// TIA Portal project "Pick and Place (Basic)" (V16)
// Vorlageprojekt für das Buch mit Zielsystem S7-1200

(* hardware
DEVICE "S7-1200-Station_1"  S7-1200 Station
   slot 0: "Baugruppenträger_0"  Rack  V1.0
   slot 1: "PLC_1"  CPU 1211C DC/DC/DC  6ES7 211-1AE40-0XB0  V4.1
*)

// ===== PLC "PLC_1"  CPU 1211C DC/DC/DC =====

VAR_GLOBAL   // PLC tag table "Standard-Variablentabelle"
   "Start" AT %I10.0 : Bool;
   "Stop" AT %I10.1 : Bool;
   "Item at entry" AT %I10.2 : Bool;
   "Item at exit" AT %I10.3 : Bool;
   "Moving X" AT %I10.4 : Bool;
   "Moving Z" AT %I10.5 : Bool;
   "Item detected" AT %I10.6 : Bool;
   "X1" AT %M1.0 : Bool;
   "X2" AT %M1.1 : Bool;
   "X3" AT %M1.2 : Bool;
   "X4" AT %M1.3 : Bool;
   "X5" AT %M1.4 : Bool;
   "X6" AT %M1.5 : Bool;
   "Entry Conveyor" AT %Q10.0 : Bool;
   "Exit Conveyor" AT %Q10.1 : Bool;
   "Move X" AT %Q10.2 : Bool;
   "Move Z" AT %Q10.3 : Bool;
   "Grab" AT %Q10.4 : Bool;
   "X7" AT %M1.6 : Bool;
   "X8" AT %M1.7 : Bool;
END_VAR

// folder: System blocks/Program resources

DATA_BLOCK "T1"   // DB1
{ S7_Optimized_Access := 'TRUE' }
AUTHOR : Simatic
FAMILY : IEC
NAME : IEC_TMR
VERSION : 1.0
// stored: InstanceOfName IEC_TIMER
"IEC_TIMER"
BEGIN
END_DATA_BLOCK

DATA_BLOCK "T2"   // DB2
{ S7_Optimized_Access := 'TRUE' }
AUTHOR : Simatic
FAMILY : IEC
NAME : IEC_TMR
VERSION : 1.0
// stored: InstanceOfName IEC_TIMER
"IEC_TIMER"
BEGIN
END_DATA_BLOCK

// folder: (top level)

FUNCTION "MHJ-PLC-Lab-Function-S71200" : Void   // FC9000, SCL
{ S7_Optimized_Access := 'TRUE' }
VERSION : 0.1
   VAR_TEMP
      rdTimeReturn : Int;
      outputTime : DTL;
      SyncVal : Byte;
      forVal : Int;
      forVal_2 : Int;
      Value : Byte;
   END_VAR
   VAR CONSTANT
      CompVal : Byte := 16#34;
      Value_01 : Byte := 16#11;
      Value_01_DW : DWord := 16#A165_D992;
      Value_02_DW : DWord := 16#58BE_4401;
   END_VAR
BEGIN

   #Value:=PEEK(area := 16#82,
        dbNumber := 0,
        byteOffset := 511);
   #Value := #Value + 1;

   POKE(area := 16#82,
        dbNumber := 0,
        byteOffset := 511,
        value := #Value);

   POKE(area:=16#81,
        dbNumber:=0,
        byteOffset:=1016,
        value:=#Value_01_DW);
   POKE(area := 16#81,
        dbNumber := 0,
        byteOffset := 1020,
        value := #Value_02_DW);

   POKE(area := 16#81,
        dbNumber := 0,
        byteOffset := 511,
        value := B#16#00);

   FOR #forVal := 0 TO 120 DO
       FOR #forVal_2:=0 TO 10 DO
           #rdTimeReturn:=RD_SYS_T(#outputTime);
           #rdTimeReturn := WR_SYS_T(#outputTime);
           #rdTimeReturn := RD_SYS_T(#outputTime);
           #rdTimeReturn := WR_SYS_T(#outputTime);
       END_FOR;
       #SyncVal:= PEEK(area := 16#81,
                      dbNumber := 0,
                      byteOffset := 511);
       IF #SyncVal = #CompVal THEN
          GOTO M_1;
       END_IF;
   END_FOR;
   RETURN;

   M_1:
   POKE(area := 16#81,
        dbNumber := 0,
        byteOffset := 511,
        value := B#16#0);
END_FUNCTION

ORGANIZATION_BLOCK "Main"   // OB1, LAD, ProgramCycle
TITLE = "Main Program Sweep (Cycle)"
{ S7_Optimized_Access := 'TRUE' }
VERSION : 0.1
   VAR_INPUT
      Initial_Call : Bool;   // Initial call of this OB
      Remanence : Bool;   // =True, if remanent data are available
   END_VAR
   VAR_TEMP   // added for the SCL form of the ladder/FBD networks
      _w1 : Bool;
   END_VAR
BEGIN

REGION Network 1: Konnektierungsbaustein für PLC-Lab
   // Im Netzwerk 1 wird der Konnektierungsbaustein für PLC-Lab aufgerufen.
   // Dieser Aufruf darf nicht entfernt werden!
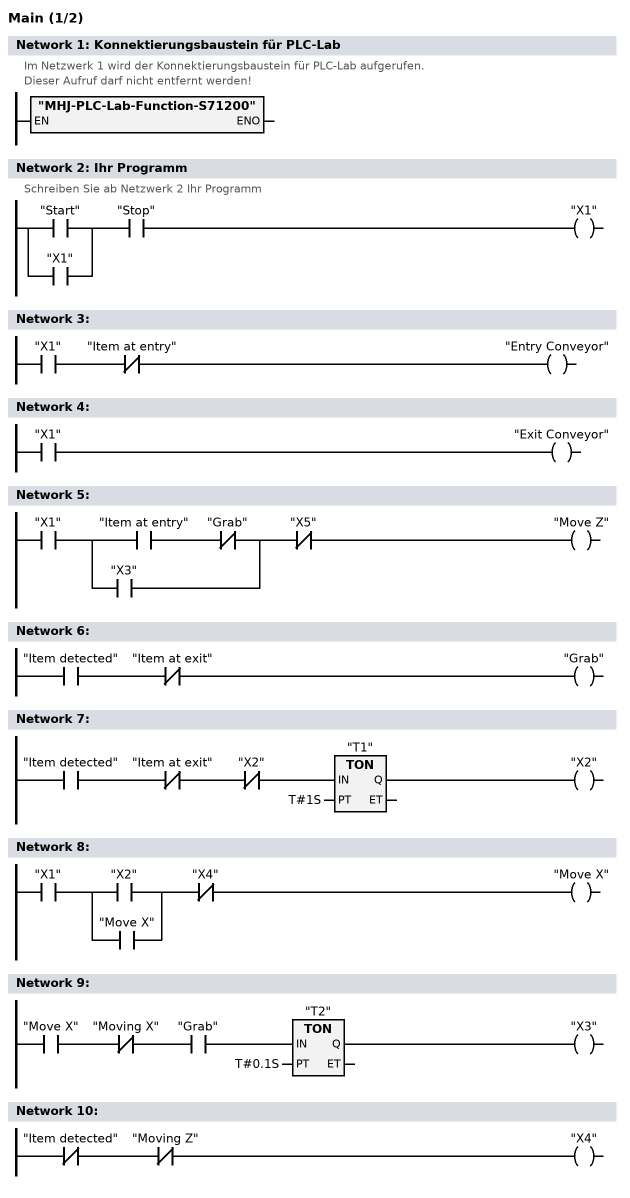
   RUNG wire#powerrail
      "MHJ-PLC-Lab-Function-S71200"()
   END_RUNG
   // the same network as SCL:
   "MHJ-PLC-Lab-Function-S71200"();
END_REGION

REGION Network 2: Ihr Programm
   // Schreiben Sie ab Netzwerk 2 Ihr Programm
   RUNG wire#powerrail
      Contact( "Start" )
      wire#w1
      Contact( "Stop" )
      Coil( "X1" )
   END_RUNG
   RUNG wire#powerrail
      Contact( "X1" )
   END_RUNG wire#w1
   // the same network as SCL:
   "X1" := ("Start" OR "X1") AND "Stop";
END_REGION

REGION Network 3
   RUNG wire#powerrail
      Contact( "X1" )
      I_Contact( "Item at entry" )
      Coil( "Entry Conveyor" )
   END_RUNG
   // the same network as SCL:
   "Entry Conveyor" := "X1" AND NOT "Item at entry";
END_REGION

REGION Network 4
   RUNG wire#powerrail
      Contact( "X1" )
      Coil( "Exit Conveyor" )
   END_RUNG
   // the same network as SCL:
   "Exit Conveyor" := "X1";
END_REGION

REGION Network 5
   RUNG wire#powerrail
      Contact( "X1" )
      wire#w1
      Contact( "Item at entry" )
      I_Contact( "Grab" )
      wire#w2
      I_Contact( "X5" )
      Coil( "Move Z" )
   END_RUNG
   RUNG wire#w1
      Contact( "X3" )
   END_RUNG wire#w2
   // the same network as SCL:
   "Move Z" := "X1" AND (("Item at entry" AND NOT "Grab") OR "X3") AND NOT "X5";
END_REGION

REGION Network 6
   RUNG wire#powerrail
      Contact( "Item detected" )
      I_Contact( "Item at exit" )
      Coil( "Grab" )
   END_RUNG
   // the same network as SCL:
   "Grab" := "Item detected" AND NOT "Item at exit";
END_REGION

REGION Network 7
   "T1".TON(IN := "Item detected" AND NOT "Item at exit" AND NOT "X2", PT := T#1S);
   "X2" := "T1".Q;
END_REGION

REGION Network 8
   RUNG wire#powerrail
      Contact( "X1" )
      wire#w1
      Contact( "X2" )
      wire#w2
      I_Contact( "X4" )
      Coil( "Move X" )
   END_RUNG
   RUNG wire#w1
      Contact( "Move X" )
   END_RUNG wire#w2
   // the same network as SCL:
   "Move X" := "X1" AND ("X2" OR "Move X") AND NOT "X4";
END_REGION

REGION Network 9
   "T2".TON(IN := "Move X" AND NOT "Moving X" AND "Grab", PT := T#0.1S);
   "X3" := "T2".Q;
END_REGION

REGION Network 10
   RUNG wire#powerrail
      I_Contact( "Item detected" )
      I_Contact( "Moving Z" )
      Coil( "X4" )
   END_RUNG
   // the same network as SCL:
   "X4" := NOT "Item detected" AND NOT "Moving Z";
END_REGION

REGION Network 11
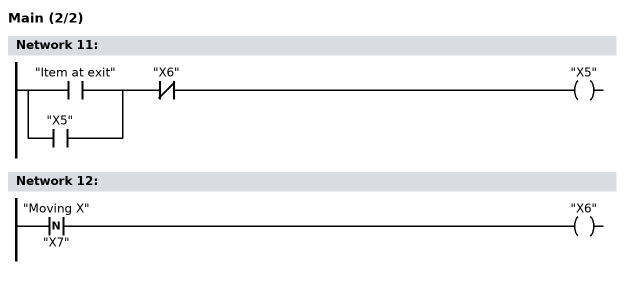
   RUNG wire#powerrail
      Contact( "Item at exit" )
      wire#w1
      I_Contact( "X6" )
      Coil( "X5" )
   END_RUNG
   RUNG wire#powerrail
      Contact( "X5" )
   END_RUNG wire#w1
   // the same network as SCL:
   "X5" := ("Item at exit" OR "X5") AND NOT "X6";
END_REGION

REGION Network 12
   RUNG wire#powerrail
      N_Contact(operand := "Moving X", bit := "X7")
      Coil( "X6" )
   END_RUNG
   // the same network as SCL:
   #_w1 := NOT "Moving X" AND "X7";   // falling edge of "Moving X"
   "X7" := "Moving X";
   "X6" := #_w1;
END_REGION
END_ORGANIZATION_BLOCK